Staubli VAL3: findValue.pgx

public program findValue(string& x_sItem[], num& x_nValue[], num& x_nValue1[])
  local num l_nSize
  local string l_sItem
begin
  //
  // find one item in the list
  //
  call getSize(l_nSize)
  for i=0 to l_nSize
    call get(l_sItem,i)
    if l_sItem==x_sItem
      call getValue(x_nValue,i,x_nValue1)
      return
      //go back
    endIf
  endFor
end
